# EPICS autosave request: ADApp/Db/NDCodec_settings.req
$(P)$(R)Mode
$(P)$(R)Compressor
$(P)$(R)JPEGQuality
$(P)$(R)BloscCompressor
$(P)$(R)BloscCLevel
$(P)$(R)BloscShuffle
$(P)$(R)BloscNumThreads
$(P)$(R)LZ4HDF5BlockSize
file "NDPluginBase_settings.req", P=$(P), R=$(R)
